FUNCTION_BLOCK FB_Alimentador_SFC // EXTENDS FB_Module_SFC
VAR_INPUT
	IC: BOOL;
	Execute: BOOL;
	Ack: BOOL;
END_VAR
VAR_OUTPUT
	Ready: BOOL;
	Failure: BOOL;
	Done: BOOL;
END_VAR

VAR_INPUT
	TK_1: TIME;					// Temporizador empujador tapa
	k1: BOOL; 					// Sensor de empujador tapa delante
END_VAR
VAR_OUTPUT
	K_1: BOOL; (* Actuador de empujador tapa avanza *)
	FM : BOOL; 
END_VAR
VAR
	tm: S_Timeouts;
END_VAR

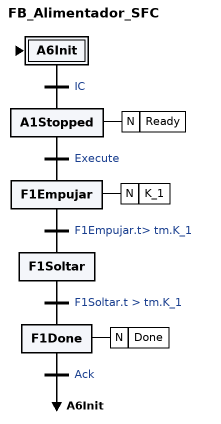
INITIAL_STEP A6Init:
END_STEP
TRANSITION FROM A6Init TO A1Stopped
    := IC;
END_TRANSITION
STEP A1Stopped:
    Ready(N);
END_STEP
TRANSITION FROM A1Stopped TO F1Empujar
    := Execute;
END_TRANSITION
STEP F1Empujar:
    K_1(N);
END_STEP
TRANSITION FROM F1Empujar TO F1Soltar
    := F1Empujar.t> tm.K_1;
END_TRANSITION
STEP F1Soltar:
END_STEP
TRANSITION FROM F1Soltar TO F1Done
    := F1Soltar.t > tm.K_1;
END_TRANSITION
STEP F1Done:
    Done(N);
END_STEP
TRANSITION FROM F1Done TO A6Init
    := Ack;
END_TRANSITION

END_FUNCTION_BLOCK

(* stored: Version 1.1.0.1, ProductVersion 3.1.4024.11
   POU FB_Alimentador_SFC: Id {25ad7b61-92b1-41db-8b65-16e3fd2054f3}, SpecialFunc None *)
